TYPE orderHmiCommands_TypeStruct :
STRUCT
	
	changeOrder				: BOOL;
	resetUpperLevelCounter	: BOOL;	(*Reset upper level sheet counter*)
	resetLowerLevelCounter	: BOOL;	(*Reset lower level sheet counter*)

END_STRUCT
END_TYPE

(* stored: Version 1.1.0.1
   DUT orderHmiCommands_TypeStruct: Id {d5da5354-4b4f-4785-aaaf-c533bf2b051a} *)
